{attribute 'GeneratedUsingTerminal: EL3773-0000-0016'}
{attribute addProperty BoxType "EL3773-0000-0016"}
{attribute addProperty Id "U3_STATUSAT %I*U3_STATUS_B07533568"}
{attribute addProperty CRC "738312571"}
{attribute addProperty Size "8"}
TYPE L3_Voltage_Status_2C01C17B EXTENDS InputBase_8311D824 :
STRUCT
	{attribute addProperty Name "U3_STATUS"}
	U3_STATUS AT %I* : U3_STATUS_B0753356;
END_STRUCT
END_TYPE

(* stored: Version 1.2.0.0, ProductVersion 3.1.4024.9
   DUT L3_Voltage_Status_2C01C17B: Id {89e9e62e-3847-40ac-a969-d429b586a032} *)
